(*
SPDX-FileCopyrightText: © 2026 Oleksandr Tiutyk <trofimich@gmail.com>
SPDX-License-Identifier: MIT
License: https://opensource.org/license/mit
*)

{attribute 'no_explicit_call' := 'do not call this function block directly'} 
FUNCTION_BLOCK SetErrorAndStopExceptionHandlingPolicy EXTENDS Object IMPLEMENTS IExceptionHandlingPolicy
VAR
	{attribute 'hide'} 
	_ClassName : STRING := __POUNAME();
END_VAR

{attribute 'monitoring' := 'call'}
PROPERTY ClassName : REFERENCE TO STRING
GET
ClassName REF= _ClassName;
END_GET
END_PROPERTY

METHOD HandleException : EXCEPTION_REACTION
VAR_INPUT
	exception : IReadOnlyException;
	handlingObject : IObject;
END_VAR
VAR_IN_OUT CONSTANT
	failedMethodName : STRING(255);
END_VAR
HandleException := EXCEPTION_REACTION.SET_ERROR_AND_STOP;
END_METHOD

{attribute 'monitoring' := 'call'}
PROPERTY NamespaceName : REFERENCE TO STRING
GET
NamespaceName REF= CurrentNamespace.Name;
END_GET
END_PROPERTY

{attribute 'monitoring' := 'call'}
PROPERTY SelfSize : ULINT
GET
SelfSize := XSIZEOF(THIS^);
END_GET
END_PROPERTY

END_FUNCTION_BLOCK

(* stored: Version 1.1.0.1
   POU SetErrorAndStopExceptionHandlingPolicy: Id {147e24e0-52f1-4730-b874-817dcb4f0d6e}, SpecialFunc None
   Property ClassName: Id {be05c405-8b13-4da0-9af2-b990288b8304}
   Get Get: Id {8d8b46db-822b-4de2-aa85-ad0ff159a192}
   Method HandleException: Id {8f660e0b-0432-46e5-a732-fed998bb6ec7}
   Property NamespaceName: Id {71485a56-6739-4b28-8d83-b88a603a6250}
   Get Get: Id {8337be40-ebdf-4028-be41-eb05a3e8735e}
   Property SelfSize: Id {4af0138b-52f1-442e-b6ca-187c312846e0}
   Get Get: Id {2907f3f1-dafe-4c50-a54b-524d25a63c58} *)
